// TIA Portal V20 export
DATA_BLOCK "ControlNodes"   // DB70
{ DB_Accessible_From_OPC_UA := 'FALSE' }
AUTHOR : ERsystem_FA2_DH. Kim
// stored: DBAccessibleFromOPCUA false, DBAccessibleFromWebserver false, MemoryReserve 100, Namespace Unit1.Em1
   VAR
      em { ExternalWritable := 'False'} : "LAF_typeEmControlNode";
      cm : Struct
         Interlock : Struct
            unwinderBtmAxisB : "LER_typeAxisInterlock";
            airShaftBtmOnOff { S7_SetPoint := 'True'} : "LER_typeTwoWayActInterlock";
         END_STRUCT;
         command : Struct
            unwinderBtmAxisB : "LER_typeAxisCommand";
            airShaftBtmOnOff { S7_SetPoint := 'True'} : "LER_typeTwoWayActCommand";
         END_STRUCT;
         softCam : "Unit1.type_emRelations_em1_SoftCam";
         brakeTest : Struct
            UnwinderBtmAxisB : "LER_typeBrakeTestEmControlNoeds";
         END_STRUCT;
      END_STRUCT;
      citiMap : "LER_OEM_Data";
      sepaUnwinderBtm : Struct
         jobs : "LAF_typeJobs";
         sequence { S7_SetPoint := 'True'} : "LAF_typeSequence";
         "step" { S7_SetPoint := 'True'} : "LER_typeStep";
         jobInterface : Struct
            reqAutoSplice : Bool;
            busyAutoSplice : Bool;
            doneAutoSplice : Bool;
         END_STRUCT;
         preOperationCheck : Struct
            home : Bool;
            homeSummary : Bool;
            Bool3 : Bool;
            Bool4 : Bool;
            Bool5 : Bool;
            Bool6 : Bool;
            Bool7 : Bool;
            Bool8 : Bool;
            Bool9 : Bool;
            Bool10 : Bool;
            Bool11 : Bool;
            Bool12 : Bool;
            Bool13 : Bool;
            Bool14 : Bool;
            Bool15 : Bool;
            Bool16 : Bool;
            Bool17 : Bool;
            Bool18 : Bool;
            Bool19 : Bool;
            Bool20 : Bool;
         END_STRUCT;
      END_STRUCT;
      emRelations : Struct
         em2 : Struct
            reqRewind : Bool;
            reqEm0To1LinkChg : Bool;
            reqEm1To0LinkChg : Bool;
            busyAutoSplice : Bool;
            doneAutoSplice : Bool;
         END_STRUCT;
         em3 : Struct
            cmStatus : Struct
               dancerRegulator { ExternalWritable := 'False'} : "LBC_typeTwoWayActuatorControlNodeMonitoring";
               dancerEncoder { ExternalWritable := 'False'} : "LBC_typeAnalogInputControlNodeMonitoring";
            END_STRUCT;
         END_STRUCT;
      END_STRUCT;
      motionRelations : Struct
         commands : Struct
            null : Bool;
         END_STRUCT;
         monitoring : Struct
            null : Bool;
         END_STRUCT;
         config : Struct
            null : Bool;
         END_STRUCT;
      END_STRUCT;
      cmBtmDirectionCheckSensor { S7_SetPoint := 'True'} : "LBC_typeDigitalSignalControlNode";
      cmRadiusMeasureBtm { ExternalAccessible := 'False'; ExternalVisible := 'False'; ExternalWritable := 'False'} : "LBC_typeAnalogInputControlNode";
      cmRadiusMeasure { ExternalWritable := 'False'} : "LER_typeRadiusMeasureControlNode";
      cmUnwinderBtmAxisB { ExternalAccessible := 'False'; ExternalVisible := 'False'; ExternalWritable := 'False'; S7_SetPoint := 'True'} : "LBC_typeAxis64PosControlNode";
      cmAirShaftBtmOnOff { ExternalAccessible := 'False'; ExternalVisible := 'False'; ExternalWritable := 'False'; S7_SetPoint := 'True'} : "LBC_typeTwoWayActuatorControlNode";
      cmEpcBtm { ExternalAccessible := 'False'; ExternalVisible := 'False'; ExternalWritable := 'False'} : "LER_typeCON600ControlNode";
   END_VAR
BEGIN
   em.commands.enable := FALSE;
   em.commands.acknowledge := FALSE;
   em.commands.disableAlarms := FALSE;
   em.commands.activateSimulation := FALSE;
   em.commands.home := FALSE;
   em.commands.moveToInitialPosition := FALSE;
   em.commands.directModeControl.current := 2;
   em.commands.directModeControl.production := FALSE;
   em.commands.directModeControl.maintenance := TRUE;
   em.commands.directModeControl.manual := FALSE;
   em.commands.directModeControl.nomode := FALSE;
   em.commands.directModeControl.sleep := FALSE;
   em.commands.directModeControl.deepsleep := FALSE;
   em.commands.directModeControl.userMode04 := FALSE;
   em.commands.directModeControl.userMode05 := FALSE;
   em.commands.directModeControl.userMode06 := FALSE;
   em.commands.directModeControl.userMode07 := FALSE;
   em.commands.directModeControl.userMode08 := FALSE;
   em.commands.directModeControl.userMode09 := FALSE;
   em.commands.directModeControl.userMode10 := FALSE;
   em.commands.directModeControl.userMode11 := FALSE;
   em.commands.directModeControl.userMode12 := FALSE;
   em.commands.directModeControl.userMode13 := FALSE;
   em.commands.directStateControl.current := 2;
   em.commands.directStateControl.clearing := FALSE;
   em.commands.directStateControl.stopped := TRUE;
   em.commands.directStateControl.starting := FALSE;
   em.commands.directStateControl.idle := FALSE;
   em.commands.directStateControl.suspended := FALSE;
   em.commands.directStateControl.execute := FALSE;
   em.commands.directStateControl.stopping := FALSE;
   em.commands.directStateControl.aborting := FALSE;
   em.commands.directStateControl.aborted := FALSE;
   em.commands.directStateControl.holding := FALSE;
   em.commands.directStateControl.held := FALSE;
   em.commands.directStateControl.unholding := FALSE;
   em.commands.directStateControl.suspending := FALSE;
   em.commands.directStateControl.unsuspending := FALSE;
   em.commands.directStateControl.resetting := FALSE;
   em.commands.directStateControl.completing := FALSE;
   em.commands.directStateControl.complete := FALSE;
   em.status.enabled := TRUE;
   em.status.acknowledgeActive := FALSE;
   em.status.alarmsDisabled := FALSE;
   em.status.simulationActive := FALSE;
   em.status.safetyReleased := TRUE;
   em.status.initialized := FALSE;
   em.status.homed := FALSE;
   em.status.safeState := TRUE;
   em.status.stateComplete := TRUE;
   // sepaUnwinderBtm."step".action1[101] : Step[101] : JOB[1] Condition
   // sepaUnwinderBtm."step".action1[110] : Step[110] : Air Shaft Work
   // sepaUnwinderBtm."step".action1[120] : Step[120] : EPC Mode Check
   // sepaUnwinderBtm."step".action1[180] : Step[180] : Unwinder B-Axis Dancer Angle Adjust
   // sepaUnwinderBtm."step".action1[190] : Step[190] : Job [1] Step End
   // sepaUnwinderBtm."step".action1[201] : Step[201] : JOB[2] Condition
   // sepaUnwinderBtm."step".action1[280] : Step[280] : Unwinder B-Axis Unwinding [Motion]
   // sepaUnwinderBtm."step".action1[290] : Step[290] : Job[2] Step End
   // sepaUnwinderBtm."step".action1[301] : Step[301] : JOB[3] Condition
   // sepaUnwinderBtm."step".action1[380] : Step[380] : Unwinder B-Axis Stop [Motion]
   // sepaUnwinderBtm."step".action1[390] : Step[390] : Job[3] Step End
   // sepaUnwinderBtm."step".action1[401] : Step[401] : JOB[4] Condition
   // sepaUnwinderBtm."step".action1[480] : Step[480] : Unwinder B-Axis Rewinding
   // sepaUnwinderBtm."step".action1[490] : Step[490] : Job[4] Step End
   // sepaUnwinderBtm."step".transition1[101] : Step[101] : JOB[1] Condition
   // sepaUnwinderBtm."step".transition1[110] : Step[110] : Air Shaft Work
   // sepaUnwinderBtm."step".transition1[120] : Step[120] : EPC Mode Check
   // sepaUnwinderBtm."step".transition1[180] : Step[180] : Unwinder B-Axis Dancer Angle Adjust
   // sepaUnwinderBtm."step".transition1[190] : Step[190] : Job [1] Step End
   // sepaUnwinderBtm."step".transition1[201] : Step[201] : JOB[2] Condition
   // sepaUnwinderBtm."step".transition1[280] : Step[280] : Unwinder B-Axis Unwinding [Motion]
   // sepaUnwinderBtm."step".transition1[290] : Step[290] : Job[2] Step End
   // sepaUnwinderBtm."step".transition1[301] : Step[301] : JOB[3] Condition
   // sepaUnwinderBtm."step".transition1[380] : Step[380] : Unwinder B-Axis Stop [Motion]
   // sepaUnwinderBtm."step".transition1[390] : Step[390] : Job[3] Step End
   // sepaUnwinderBtm."step".transition1[401] : Step[401] : JOB[4] Condition
   // sepaUnwinderBtm."step".transition1[480] : Step[480] : Unwinder B-Axis Rewinding
   // sepaUnwinderBtm."step".transition1[490] : Step[490] : Job[4] Step End
   cmBtmDirectionCheckSensor.commands.reset := FALSE;
   cmBtmDirectionCheckSensor.commands.simulation := FALSE;
   cmBtmDirectionCheckSensor.commands.quality := TRUE;
   cmRadiusMeasureBtm.commands.simulation := FALSE;
   cmRadiusMeasureBtm.commands.reset := FALSE;
   cmRadiusMeasureBtm.commands.quality := TRUE;
   cmRadiusMeasureBtm.monitoring.valid := FALSE;
   cmRadiusMeasureBtm.monitoring.busy := FALSE;
   cmRadiusMeasureBtm.monitoring.error := TRUE;
   cmRadiusMeasureBtm.monitoring.status := 16#8405;
   cmRadiusMeasureBtm.monitoring.processValue := 0.0;
   cmRadiusMeasureBtm.monitoring.limitHigh2 := FALSE;
   cmRadiusMeasureBtm.monitoring.limitHigh1 := FALSE;
   cmRadiusMeasureBtm.monitoring.limitLow1 := TRUE;
   cmRadiusMeasureBtm.monitoring.limitLow2 := TRUE;
   cmRadiusMeasureBtm.monitoring.maxValueReached := FALSE;
   cmRadiusMeasureBtm.monitoring.minValueReached := TRUE;
   cmRadiusMeasure.commands.ZeroSet := FALSE;
   cmRadiusMeasure.commands.Reset := FALSE;
   cmRadiusMeasure.monitoring.Radius := 0.0;
   cmRadiusMeasure.monitoring.Diameter := 0.0;
   cmAirShaftBtmOnOff.commands.commandHomePos := FALSE;
   cmAirShaftBtmOnOff.commands.commandWorkPos := FALSE;
   cmAirShaftBtmOnOff.commands.reset := FALSE;
END_DATA_BLOCK
